# EPICS substitutions: rcsRfIoc/rcsRfIocApp/Db/user.substitutions
# Example substitutions file

file "db/dbExample1.db" {
    { user = "RCS" }
}

file db/dbExample2.db {
    pattern { user, no, scan }
        { "RCS", 1, "1 second" }
        { "RCS", 2, "2 second" }
        { "RCS", 3, "5 second" }
}
